FUNCTION_BLOCK FB_Station_Disable EXTENDS FB_CH_Object
VAR

	ipStation : I_XP_Station_PLC;
END_VAR

METHOD FB_init : BOOL
VAR_INPUT
	bInitRetains : BOOL; // if TRUE, the retain variables are initialized (warm start / cold start)
	bInCopyCode : BOOL;  // if TRUE, the instance afterwards gets moved into the copy code (online change)
	
	ipStation : I_XP_Station_PLC;
	
END_VAR
VAR
	fbGetCurTaskIdx  : GETCURTASKINDEX;
END_VAR
THIS^.ipStation := ipStation;
END_METHOD

METHOD Update : HRESULT
VAR
	refPlanarTrack : REFERENCE TO MC_PlanarTrack;
END_VAR

VAR_INST
	nSeq : UINT;
	fbFeedback : MC_PlanarFeedback;
	fbTon : TON;
	ipMoverInStation : I_XP_Mover_PLC;
END_VAR
IF ipStation = 0 THEN
	RETURN; // ERROR
END_IF

IF ipStation.System.Disabled THEN
	nSeq := 0;
END_IF

ipStation.SimulationStop();

CASE nSeq OF 

	0: //wait for mover
		IF ipStation.MoversInPlace THEN
			ipMoverInStation := ipStation.MoversInQueue[0];
			nSeq := 1;
		END_IF
		
	1: //disable
		ipMoverInStation.PlanarMover.Disable(fbFeedback);
		nSeq := 2;				

	2: // wait until disable is finish
		IF fbFeedback.Done THEN
			fbTon.IN := FALSE;
			nSeq := 3;	
		END_IF
		
	3: //Delay 5s
		fbTon.IN := TRUE;
		IF fbTon.q THEN
			nSeq := 4;	
		END_IF			

	4: //enable
		ipMoverInStation.PlanarMover.Enable(fbFeedback);
		nSeq := 5;				

	5: // wait until enable is finish
		IF fbFeedback.Done THEN
			fbTon.IN := FALSE;
			nSeq := 6;	
		END_IF
		
	6: //join Track
		refPlanarTrack REF= ipStation.AccocietedTrack.PlanarTrack;
		ipMoverInStation.PlanarMover.JoinTrack(	commandFeedback	:= fbFeedback, 
												targetTrack		:= refPlanarTrack, 
												constraint		:= ipMoverInStation.DynConstraint, 
												options			:= 0);
		nSeq := 7;				

	7: // wait until enable is finish
		IF fbFeedback.Done THEN
			fbTon.IN := FALSE;
			nSeq := 8;	
		END_IF
		
	8: // send movers away
		ipStation.SendMoversToStation(MAIN.G_WorkBench);
		nSeq := 0;	
	
END_CASE
fbFeedback.Update();
fbTon(PT:= T#5S);
END_METHOD

END_FUNCTION_BLOCK

(* stored: Version 1.1.0.1, ProductVersion 3.1.4024.12
   POU FB_Station_Disable: Id {f250b27e-a3a3-4f8c-a728-76a9ef965b85}, SpecialFunc None
   Method FB_init: Id {fcb0a98d-d756-49b7-8bce-33c65cdfba9e}
   Method Update: Id {109ef4a0-0354-43ed-b4f8-08e59b74708c} *)
